// TIA Portal V18 export
FUNCTION_BLOCK "Runtime"   // FB124, LAD
{ S7_Optimized_Access := 'TRUE' }
// Written By Kristopher Gimenez March 3rd,2023
// 
// This block and its DB will perform a runtime counter and outputs total runtime in Hours, Minutes and Seconds
// stored: AutoNumber false, MemoryReserve 100, SetENOAutomatically false
   VAR_INPUT
      Start : Bool;
      Reset : Bool;
      NewHours : DInt;
      NewMins : DInt;
      NewSeconds : DInt;
   END_VAR
   VAR_OUTPUT
      TotalTime : DInt;
      TotHours : DInt;
      TotMins : DInt;
      TotSeconds : DInt;
      CurrentTime : DInt;   // Current Time in Seconds
      CurHours : DInt;
      CurMins : DInt;
      CurSeconds : DInt;
   END_VAR
   VAR
      StartTrig : Bool;
      StartTime : DInt;
      Runtime_TONR { S7_SetPoint := 'True'} : TONR_TIME;
      TimerReset { ExternalAccessible := 'False'; ExternalVisible := 'False'; ExternalWritable := 'False'} : Bool;
      CurrentIECTime : Time;
      NewTime : DInt;   // New Time in seconds to reset to base on inputs
   END_VAR
   VAR_TEMP
      TempDInt : DInt;
      NewHoursInSec : DInt;
      NewMinsInSec : DInt;
   END_VAR
   VAR_TEMP   // added for the SCL form of the ladder/FBD networks
      _w1 : Bool;
   END_VAR
BEGIN

REGION Network 1: Start
   // When Starting store Total as Start Value
   // Reset Current Runtime
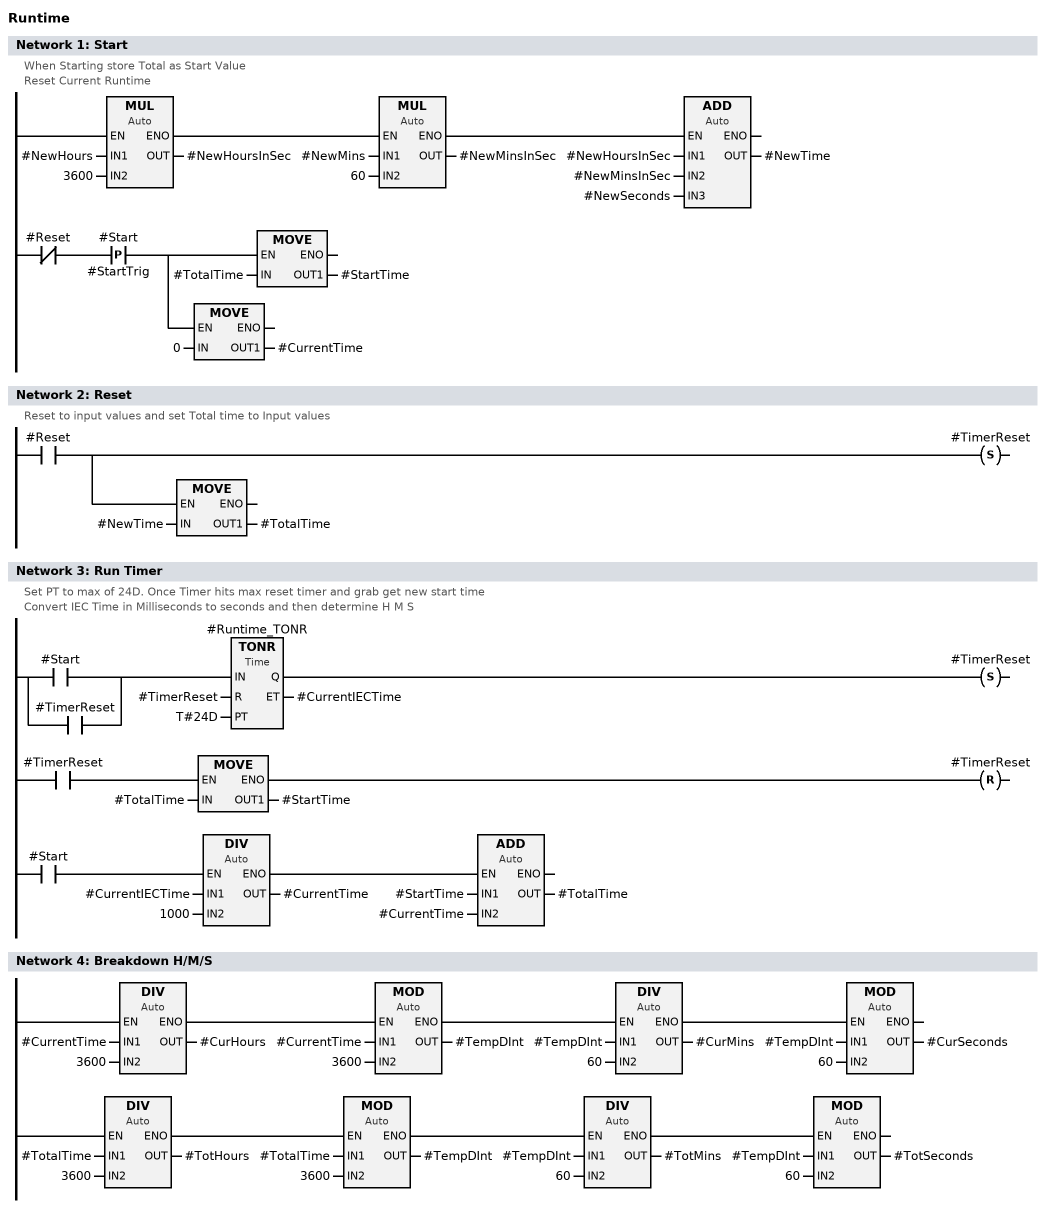
   RUNG wire#powerrail
      Mul(in1 := #NewHours, in2 := 3600, out => #NewHoursInSec)
      Mul(in1 := #NewMins, in2 := 60, out => #NewMinsInSec)
      Add(in1 := #NewHoursInSec, in2 := #NewMinsInSec, in3 := #NewSeconds, out => #NewTime)
   END_RUNG
   RUNG wire#powerrail
      I_Contact( #Reset )
      P_Contact(operand := #Start, bit := #StartTrig)
      wire#w1
      Move(in := #TotalTime, out1 => #StartTime)
   END_RUNG
   RUNG wire#w1
      Move(in := 0, out1 => #CurrentTime)
   END_RUNG
   // the same network as SCL:
   #NewHoursInSec := #NewHours * 3600;
   #NewMinsInSec := #NewMins * 60;
   #NewTime := #NewHoursInSec + #NewMinsInSec + #NewSeconds;
   #_w1 := NOT #Reset AND #Start AND NOT #StartTrig;   // rising edge of #Start
   #StartTrig := #Start;
   IF #_w1 THEN
       #StartTime := #TotalTime;
       #CurrentTime := 0;
   END_IF;
END_REGION

REGION Network 2: Reset
   // Reset to input values and set Total time to Input values
   RUNG wire#powerrail
      Contact( #Reset )
      wire#w1
      S_Coil( #TimerReset )
   END_RUNG
   RUNG wire#w1
      Move(in := #NewTime, out1 => #TotalTime)
   END_RUNG
   // the same network as SCL:
   IF #Reset THEN
       #TimerReset := TRUE;
       #TotalTime := #NewTime;
   END_IF;
END_REGION

REGION Network 3: Run Timer
   // Set PT to max of 24D. Once Timer hits max reset timer and grab get new start time
   // Convert IEC Time in Milliseconds to seconds and then determine H M S
   RUNG wire#powerrail
      Contact( #Start )
      wire#w1
      { S7_Templates := "time_type := Time" } #Runtime_TONR.TONR(r := #TimerReset, pt := T#24D, et => #CurrentIECTime)
      S_Coil( #TimerReset )
   END_RUNG
   RUNG wire#powerrail
      Contact( #TimerReset )
   END_RUNG wire#w1
   RUNG wire#powerrail
      Contact( #TimerReset )
      Move(in := #TotalTime, out1 => #StartTime)
      R_Coil( #TimerReset )
   END_RUNG
   RUNG wire#powerrail
      Contact( #Start )
      Div(in1 := #CurrentIECTime, in2 := 1000, out => #CurrentTime)
      Add(in1 := #StartTime, in2 := #CurrentTime, out => #TotalTime)
   END_RUNG
   // the same network as SCL:
   #Runtime_TONR(IN := #Start OR #TimerReset, R := #TimerReset, PT := T#24D, ET => #CurrentIECTime);   // TONR
   IF #Runtime_TONR.Q THEN #TimerReset := TRUE; END_IF;
   IF #TimerReset THEN
       #StartTime := #TotalTime;
       #TimerReset := FALSE;
   END_IF;
   IF #Start THEN
       #CurrentTime := #CurrentIECTime / 1000;
       #TotalTime := #StartTime + #CurrentTime;
   END_IF;
END_REGION

REGION Network 4: Breakdown H/M/S
   RUNG wire#powerrail
      Div(in1 := #CurrentTime, in2 := 3600, out => #CurHours)
      Mod(in1 := #CurrentTime, in2 := 3600, out => #TempDInt)
      Div(in1 := #TempDInt, in2 := 60, out => #CurMins)
      Mod(in1 := #TempDInt, in2 := 60, out => #CurSeconds)
   END_RUNG
   RUNG wire#powerrail
      Div(in1 := #TotalTime, in2 := 3600, out => #TotHours)
      Mod(in1 := #TotalTime, in2 := 3600, out => #TempDInt)
      Div(in1 := #TempDInt, in2 := 60, out => #TotMins)
      Mod(in1 := #TempDInt, in2 := 60, out => #TotSeconds)
   END_RUNG
   // the same network as SCL:
   #CurHours := #CurrentTime / 3600;
   #TempDInt := #CurrentTime MOD 3600;
   #CurMins := #TempDInt / 60;
   #CurSeconds := #TempDInt MOD 60;
   #TotHours := #TotalTime / 3600;
   #TempDInt := #TotalTime MOD 3600;
   #TotMins := #TempDInt / 60;
   #TotSeconds := #TempDInt MOD 60;
END_REGION
END_FUNCTION_BLOCK
